{attribute addProperty BoxType "EJ1918-0000-0017"}
{attribute addProperty Id "FSOEAT %I*FSOE_314B848F567"}
{attribute addProperty CRC "726936807"}
{attribute addProperty SizeInBites "56"}
{attribute addProperty SizeInBytes "7"}
TYPE FSoE_Inputs_2B542CE7 :
STRUCT
	{attribute addProperty Name "FSOE"}
	FSOE AT %I* : FSOE_314B848F;
END_STRUCT
END_TYPE

(* stored: Version 1.2.0.0, ProductVersion 3.1.4024.9
   DUT FSoE_Inputs_2B542CE7: Id {00d4c36a-73a7-4d13-bb20-00ce75ebcca9} *)
